FUNCTION_BLOCK F_TRUNC (* truncation toward zero *)
  (* Standard: 61131-3; Classification: type conversion function *)
  (* Version 0.0, 2013-08-29, 4DIAC-IDE, 4DIAC-Consortium *)
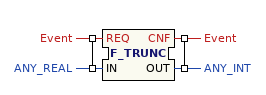
  EVENT_INPUT
    REQ WITH IN; (* Service Request *)
  END_EVENT
  EVENT_OUTPUT
    CNF WITH OUT; (* Confirmation of Requested Service *)
  END_EVENT
  VAR_INPUT
    IN : ANY_REAL; (* input value *)
  END_VAR
  VAR_OUTPUT
    OUT : ANY_INT; (* output value *)
  END_VAR
  (* Service APPLICATION/RESOURCE: truncation toward zero *)
END_FUNCTION_BLOCK
